INTERFACE ITF_Sensor2NODecoratorTest EXTENDS ITF_SensorDecoratorTest

METHOD SetContract2
VAR_INPUT
	bIN: BOOL;
END_VAR
END_METHOD

END_INTERFACE

(* stored: Version 1.1.0.1
   Itf ITF_Sensor2NODecoratorTest: Id {af78f01e-09ca-42ab-8153-e581f82e560c}
   Method SetContract2: Id {4cf85473-9fa1-43f7-af3e-def32ecc3796} *)
